FUNCTION_BLOCK GET_FEATURE_START_POINT (* Get feature start point *)
  (* Standard: 61499-2 *)
  (* Version 1.0, 14-05-12, GASR, Universidade do Estado de Santa Catarina *)
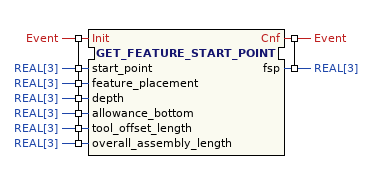
  EVENT_INPUT
    Init WITH start_point, feature_placement, depth, allowance_bottom, tool_offset_length, overall_assembly_length;
  END_EVENT
  EVENT_OUTPUT
    Cnf WITH fsp;
  END_EVENT
  VAR_INPUT
    start_point : ARRAY [0..2] OF REAL; (* Operation start point *)
    feature_placement : ARRAY [0..2] OF REAL; (* Feature local coordinate system origin *)
    depth : ARRAY [0..2] OF REAL; (* Feature depth *)
    allowance_bottom : ARRAY [0..2] OF REAL; (* Material thickness to be left uncut *)
    tool_offset_length : ARRAY [0..2] OF REAL; (* Tool blade length *)
    overall_assembly_length : ARRAY [0..2] OF REAL; (* Tool length *)
  END_VAR
  VAR_OUTPUT
    fsp : ARRAY [0..2] OF REAL; (* feature_start_point *)
  END_VAR
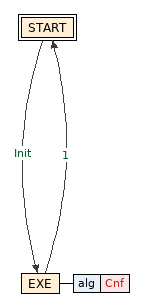
  EC_STATES
    START;
    EXE : alg -> Cnf;
  END_STATES
  EC_TRANSITIONS
    START TO EXE := Init;
    EXE TO START := 1;
  END_TRANSITIONS
  ALGORITHM alg IN Lua:
local max_depth    = depth[3] + allowance_bottom
local blade_length = overall_assembly_length - tool_offset_length
if(( start_point[1] ~= 0 ) and ( start_point[2] ~= 0 ) and ( start_point[3] ~= 0 )) then
    for i = 1, 3 do fsp[i] = start_point[i] end
else
    for i = 1, 3 do fsp[i] = feature_placement[i] end
    if( blade_length > -max_depth ) then
        fsp[3] = max_depth + feature_placement[3]
    else
        fsp[3] = -blade_length + feature_placement[3]
    end
end
print( 'start_point', fsp[1], fsp[2], fsp[3] )
print()
--Check for depth violation
if( math.abs(fsp[3] - feature_placement[3]) > blade_length ) then
    fsp[3] = -blade_length
end
if( math.abs(fsp[3] - feature_placement[3]) > max_depth ) then
    fsp[3] = -max_depth
end
  END_ALGORITHM
END_FUNCTION_BLOCK
